FUNCTION fc_Houre_To_TOD : TOD
VAR_INPUT
		IN : REAL;
END_VAR
VAR
END_VAR

fc_Houre_To_TOD := DWORD_TO_TOD(REAL_TO_DWORD(IN * 3600000));

END_FUNCTION

(* stored: Version 1.1.0.1, ProductVersion 3.1.4024.11
   POU fc_Houre_To_TOD: Id {a4f5f9ff-3198-467f-8c50-265ce4840db5}, SpecialFunc None *)
